Staubli VAL3: getPointData.pgx

public program getPointData(string x_sItem (dimensions=1), num x_nIndex (dimensions=1), point& x_pPoint (dimensions=1), bool& x_bResult (dimensions=1))
  local num i
  local num l_nResult
  local string l_sSession
begin
  // get the joint data from the specific session...
  x_bResult=false
  call saveData:getSession(l_sSession)
  // get the colletion type...
  if sSession2!=l_sSession
    // copy back
    sSession2=l_sSession
    // load the actual one
    l_nResult=pt:libLoad(saveData:sPathTraj+"POINT")
    delay(0)
  endIf
  // use the type...
  if l_nResult==0 and isDefined(pt:tTraj[x_sItem]) and size(pt:tTraj[x_sItem].tData.pPoint)>x_nIndex
    // get the JOINT DATA
    x_pPoint=pt:tTraj[x_sItem].tData.pPoint[x_nIndex]
    delay(0)
    x_bResult=true
  endIf
end
